{attribute 'qualified_only'}
VAR_GLOBAL
	Remote_Panel:  ARRAY[1..2] OF STRUCT;
END_VAR

(* stored: Version 1.1.0.1
   GVL Force: Id {5fc99bdb-2834-42a6-a55d-ad3cc17d6169} *)
